Universal Robots PolyScope program: _adminCG-PHomeToConveyor.urp

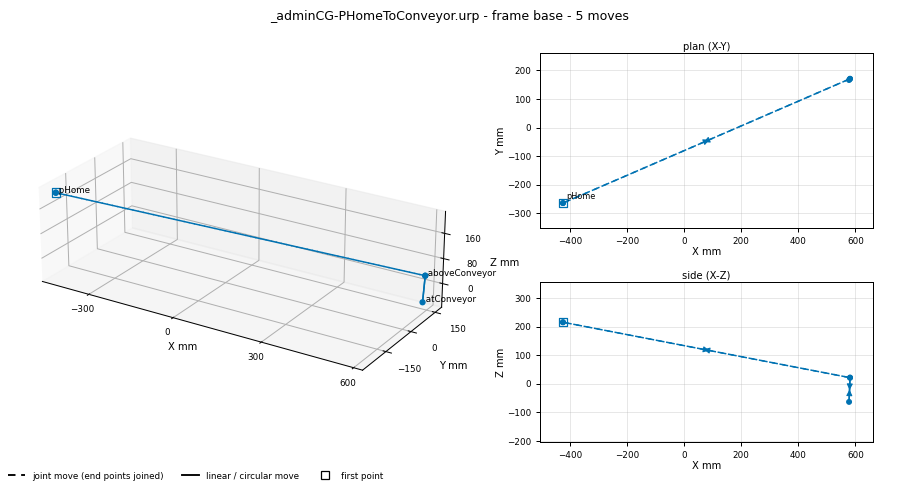
[picture p0: tool path of _adminCG-PHomeToConveyor.urp in frame base, 5 of 5 moves have a stored position in this frame; points joined in program order, loops and branches not executed]
Program _adminCG-PHomeToConveyor (installation=admin directory=/programs/THU_530PM createdIn=3.8.0.61336 lastSavedIn=3.15.8.106339 robotSerialNumber=2015350925)
Calibrated DH parameters: a=[0, -0.425, -0.39225, 0, 0, 0]; d=[0.089159, 0, 0, 0.10915, 0.09465, 0.0823]; alpha=[1.570796, 0, 0, 1.570796, -1.570796, 0]; deltaTheta=[0, 0, 0, 0, 0, 0]
Robot Program (runOnlyOnce=true)
  Set DigitalOutput pin=digital_out[0]; digitalValue=1
  Call _adminLinearIndex1
  MoveJ speed 60 deg/s, acceleration 80 deg/s^2 (useActiveTCP=true)
    Waypoint pHome: TCP in base x=-424.14 y=-264.315 z=215.866 mm, rx=-1.1973 ry=-2.8918 rz=-0.0084 rad; joints [224.999, -90.007, -90.004, -90.016, 89.259, -0.019] deg; flange x=-422.236 y=-266.361 z=431.748 mm, rx=-1.1973 ry=-2.8918 rz=-0.0084 rad
    Waypoint aboveConveyor: TCP in base x=581.102 y=170.851 z=21.809 mm, rx=2.9031 ry=-1.2001 rz=-0.0018 rad; joints [26.745, -110.225, -95.112, -64.716, 90.042, -18.335] deg; flange x=581.349 y=170.8 z=237.709 mm, rx=2.9031 ry=-1.2001 rz=-0.0018 rad
  MoveL speed 250 mm/s, acceleration 1200 mm/s^2 (useActiveTCP=true) feature=Base
    Waypoint atConveyor: TCP in base x=577.711 y=166.609 z=-63.062 mm, rx=2.9035 ry=-1.1991 rz=-0.0028 rad; joints [26.512, -115.712, -101.425, -52.94, 90.068, -18.608] deg; flange x=578.086 y=166.511 z=152.838 mm, rx=2.9035 ry=-1.1991 rz=-0.0028 rad
    Set DigitalOutput pin=digital_out[0]; digitalValue=0
    Wait Sleep waitTime=1
    Waypoint aboveConveyor: TCP in base x=581.102 y=170.851 z=21.809 mm, rx=2.9031 ry=-1.2001 rz=-0.0018 rad; joints [26.745, -110.225, -95.112, -64.716, 90.042, -18.335] deg; flange x=581.349 y=170.8 z=237.709 mm, rx=2.9031 ry=-1.2001 rz=-0.0018 rad
  MoveJ speed 60 deg/s, acceleration 80 deg/s^2 (useActiveTCP=true)
    Waypoint pHome: TCP in base x=-424.14 y=-264.315 z=215.866 mm, rx=-1.1973 ry=-2.8918 rz=-0.0084 rad; joints [224.999, -90.007, -90.004, -90.016, 89.259, -0.019] deg; flange x=-422.236 y=-266.361 z=431.748 mm, rx=-1.1973 ry=-2.8918 rz=-0.0084 rad
SubProgram  [hidden by the author, left out]
SubProgram _adminLinearIndex1 [hidden by the author, left out]
